// TIA Portal V18 export
FUNCTION_BLOCK "TD_Motor_Start_Elec"   // FB13, LAD
{ S7_Optimized_Access := 'TRUE' }
// Written BY Kristopher Gimenez January 25,2023
// This block is used to control the TD motors on an Elec HPUs
// stored: AutoNumber false, MemoryReserve 100, SetENOAutomatically false
   VAR
      TDP1FailTON { S7_SetPoint := 'True'} : TON_TIME;
      TDP2FailTON { S7_SetPoint := 'True'} : TON_TIME;
   END_VAR
BEGIN

REGION Network 1: Enable Top Drive
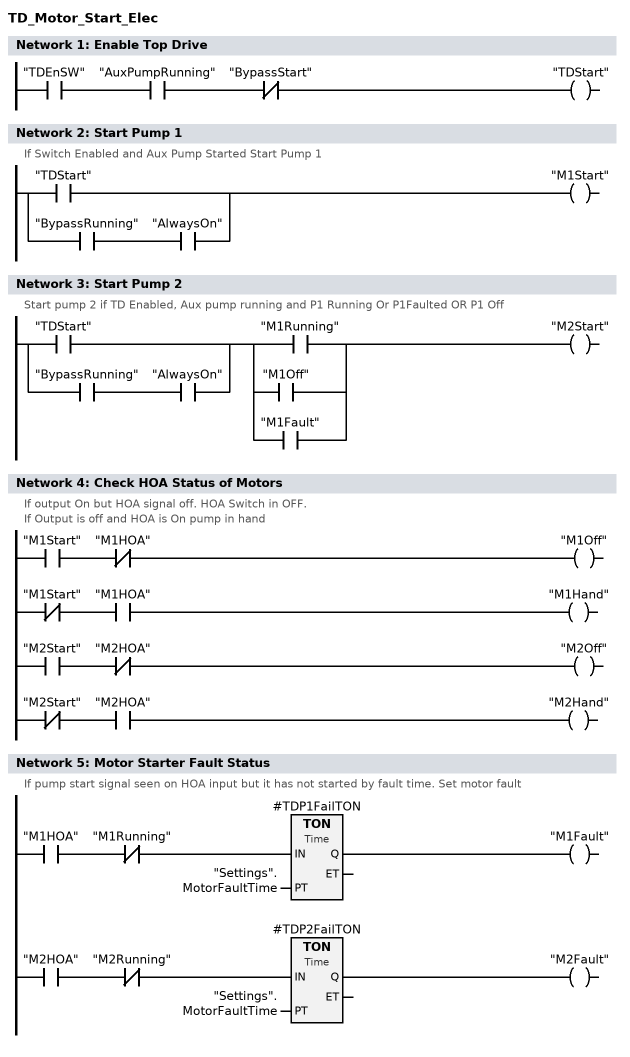
   RUNG wire#powerrail
      Contact( "TDEnSW" )
      Contact( "AuxPumpRunning" )
      I_Contact( "BypassStart" )
      Coil( "TDStart" )
   END_RUNG
   // the same network as SCL:
   "TDStart" := "TDEnSW" AND "AuxPumpRunning" AND NOT "BypassStart";
END_REGION

REGION Network 2: Start Pump 1
   // If Switch Enabled and Aux Pump Started Start Pump 1
   RUNG wire#powerrail
      Contact( "TDStart" )
      wire#w1
      Coil( "M1Start" )
   END_RUNG
   RUNG wire#powerrail
      Contact( "BypassRunning" )
      Contact( "AlwaysOn" )
   END_RUNG wire#w1
   // the same network as SCL:
   "M1Start" := "TDStart" OR ("BypassRunning" AND "AlwaysOn");
END_REGION

REGION Network 3: Start Pump 2
   // Start pump 2 if TD Enabled, Aux pump running and P1 Running Or P1Faulted OR P1 Off
   RUNG wire#powerrail
      Contact( "TDStart" )
      wire#w1
      Contact( "M1Running" )
      wire#w2
      Coil( "M2Start" )
   END_RUNG
   RUNG wire#powerrail
      Contact( "BypassRunning" )
      Contact( "AlwaysOn" )
   END_RUNG wire#w1
   RUNG wire#w1
      Contact( "M1Off" )
   END_RUNG wire#w2
   RUNG wire#w1
      Contact( "M1Fault" )
   END_RUNG wire#w2
   // the same network as SCL:
   "M2Start" := ("TDStart" OR ("BypassRunning" AND "AlwaysOn")) AND ("M1Running" OR "M1Off" OR "M1Fault");
END_REGION

REGION Network 4: Check HOA Status of Motors
   // If output On but HOA signal off. HOA Switch in OFF. 
   // If Output is off and HOA is On pump in hand
   RUNG wire#powerrail
      Contact( "M1Start" )
      I_Contact( "M1HOA" )
      Coil( "M1Off" )
   END_RUNG
   RUNG wire#powerrail
      I_Contact( "M1Start" )
      Contact( "M1HOA" )
      Coil( "M1Hand" )
   END_RUNG
   RUNG wire#powerrail
      Contact( "M2Start" )
      I_Contact( "M2HOA" )
      Coil( "M2Off" )
   END_RUNG
   RUNG wire#powerrail
      I_Contact( "M2Start" )
      Contact( "M2HOA" )
      Coil( "M2Hand" )
   END_RUNG
   // the same network as SCL:
   "M1Off" := "M1Start" AND NOT "M1HOA";
   "M1Hand" := NOT "M1Start" AND "M1HOA";
   "M2Off" := "M2Start" AND NOT "M2HOA";
   "M2Hand" := NOT "M2Start" AND "M2HOA";
END_REGION

REGION Network 5: Motor Starter Fault Status
   // If pump start signal seen on HOA input but it has not started by fault time. Set motor fault
   RUNG wire#powerrail
      Contact( "M1HOA" )
      I_Contact( "M1Running" )
      { S7_Templates := "time_type := Time" } #TDP1FailTON.TON(pt := "Settings".MotorFaultTime, et =>)
      Coil( "M1Fault" )
   END_RUNG
   RUNG wire#powerrail
      Contact( "M2HOA" )
      I_Contact( "M2Running" )
      { S7_Templates := "time_type := Time" } #TDP2FailTON.TON(pt := "Settings".MotorFaultTime, et =>)
      Coil( "M2Fault" )
   END_RUNG
   // the same network as SCL:
   #TDP1FailTON(IN := "M1HOA" AND NOT "M1Running", PT := "Settings".MotorFaultTime);   // TON
   "M1Fault" := #TDP1FailTON.Q;
   #TDP2FailTON(IN := "M2HOA" AND NOT "M2Running", PT := "Settings".MotorFaultTime);   // TON
   "M2Fault" := #TDP2FailTON.Q;
END_REGION
END_FUNCTION_BLOCK
